FUNCTION_BLOCK FB_GantryAutoCoupling
VAR_INPUT
	nGantryTol : LINT;
END_VAR
VAR_OUTPUT
	bGantryAlreadyCoupled : BOOL;
END_VAR
VAR_IN_OUT
	Master : DUT_MotionStage;
	MasterEnc : ST_RenishawAbsEnc;
	Slave : DUT_MotionStage;
	SlaveEnc : ST_RenishawAbsEnc;
	bExecuteCouple : BOOL;
	bExecuteDecouple : BOOL;
END_VAR
VAR
	gantry_diff_limit : FB_GantryDiffVirtualLimitSwitch;
	couple : MC_GEARIN;
	decouple : MC_GEAROUT;
	bInitComplete : BOOL;
	fbSetEnables : FB_SetEnables;
END_VAR

// Designate Master and SLave Axes
Master.bGantryAxis := TRUE;
Slave.bGantryAxis := TRUE;

Master.nGantryTol := nGantryTol;
Slave.nGantryTol := Master.nGantryTol;

// Activate Gantry Virtual Limit Switch
gantry_diff_limit(Penc:=MasterEnc, SEnc:=SlaveEnc, GantDiffTol:=Master.nGantryTol,
				  PLimFwd=>Master.bGantryForwardEnable, PLimBwd=>Master.bGantryBackwardEnable,
				  SLimFwd=>Slave.bGantryForwardEnable, SLimBwd=>Slave.bGantryBackwardEnable);

// Coupling Status Bit
bGantryAlreadyCoupled := Master.Axis.NcToPlc.CoupleState=1 AND Slave.Axis.NcToPlc.CoupleState=3;

fbSetEnables(stMotionStage:=Master);
fbSetEnables(stMotionStage:=Slave);

IF bGantryAlreadyCoupled THEN
	Master.bGantryForwardEnable := Master.bGantryForwardEnable AND Slave.bAllForwardEnable;
	Slave.bGantryForwardEnable := Master.bAllForwardEnable AND Slave.bGantryForwardEnable;
	
	Master.bGantryBackwardEnable := Master.bGantryBackwardEnable AND Slave.bAllBackwardEnable;
	Slave.bGantryBackwardEnable := Master.bAllBackwardEnable AND Slave.bGantryBackwardEnable;
END_IF


// Coupling states
// Auto-coupling at init and auto-reset of coupling boolean
bExecuteCouple S= NOT bInitComplete;

bExecuteCouple R= couple.Busy OR bGantryAlreadyCoupled;
couple(Master:=Master.Axis, Slave:=Slave.Axis, Execute:=bExecuteCouple);

bInitComplete S= bGantryAlreadyCoupled;

// Decoupling with auto-reset of coupling boolean
bExecuteDecouple R= decouple.Busy OR NOT bGantryAlreadyCoupled;
decouple(Slave:=Slave.Axis, Execute:=bExecuteDecouple);

END_FUNCTION_BLOCK

(* stored: Version 1.1.0.1, ProductVersion 3.1.4022.12
   POU FB_GantryAutoCoupling: Id {532dfcaf-6187-4140-aaad-e20a9bbe6b43}, SpecialFunc None *)
